// TIA Portal V18 export
TYPE "TM_Pulse_2x24_Out_PWM"
   STRUCT
      OUTPUT_VALUE : UDInt;   // Pulse Duration
      SLOT : UDInt;   // Load Value
      LD_SLOT_Bit0 : Bool;
      LD_SLOT_Bit1 : Bool;
      LD_SLOT_Bit2 : Bool;
      LD_SLOT_Bit3 : Bool;
      MODE_SLOT : Bool;
      Reserved1 : Bool;
      Reserved2 : Bool;
      Reserved3 : Bool;
      SW_ENABLE : Bool;
      TM_CTRL_DQ : Bool;
      Reserved4 : Bool;
      SET_DQA : Bool;
      SET_DQB : Bool;
      DITHER : Bool;
      Rerserved6 : Bool;
      Rerserved7 : Bool;
      RES_ERROR : Bool;
      Reserved8 : Bool;
      Reserved9 : Bool;
      Reserved10 : Bool;
      Reserved11 : Bool;
      Reserved12 : Bool;
      Reserved13 : Bool;
      Reserved14 : Bool;
      Rerserved : Byte;
   END_STRUCT;
END_TYPE
